# EPICS StreamDevice protocol: Module_12_Stream_Device/sd/sd.proto
Terminator = CR LF;

getTime{
	out "time";
	in "%s";
}
